(* IEC 61131-3 sources: drain_system/build, 2 files *)

(* ---- plc.st ---- *)
TYPE
  LOGLEVEL : (CRITICAL, WARNING, INFO, DEBUG) := INFO;
END_TYPE

FUNCTION_BLOCK LOGGER
  VAR_INPUT
    TRIG : BOOL;
    MSG : STRING;
    LEVEL : LOGLEVEL := INFO;
  END_VAR
  VAR
    TRIG0 : BOOL;
  END_VAR

  IF TRIG AND NOT TRIG0 THEN
  {{
   LogMessage(GetFbVar(LEVEL),(char*)GetFbVar(MSG, .body),GetFbVar(MSG, .len));
  }}
  END_IF;
  TRIG0:=TRIG;
END_FUNCTION_BLOCK

FUNCTION_BLOCK python_eval
  VAR_INPUT
    TRIG : BOOL;
    CODE : STRING;
  END_VAR
  VAR_OUTPUT
    ACK : BOOL;
    RESULT : STRING;
  END_VAR
  VAR
    STATE : DWORD;
    BUFFER : STRING;
    PREBUFFER : STRING;
    TRIGM1 : BOOL;
    TRIGGED : BOOL;
  END_VAR

  {extern void __PythonEvalFB(int, PYTHON_EVAL*);__PythonEvalFB(0, data__);}
END_FUNCTION_BLOCK

FUNCTION_BLOCK python_poll
  VAR_INPUT
    TRIG : BOOL;
    CODE : STRING;
  END_VAR
  VAR_OUTPUT
    ACK : BOOL;
    RESULT : STRING;
  END_VAR
  VAR
    STATE : DWORD;
    BUFFER : STRING;
    PREBUFFER : STRING;
    TRIGM1 : BOOL;
    TRIGGED : BOOL;
  END_VAR

  {extern void __PythonEvalFB(int, PYTHON_EVAL*);__PythonEvalFB(1,(PYTHON_EVAL*)(void*)data__);}
END_FUNCTION_BLOCK

FUNCTION_BLOCK python_gear
  VAR_INPUT
    N : UINT;
    TRIG : BOOL;
    CODE : STRING;
  END_VAR
  VAR_OUTPUT
    ACK : BOOL;
    RESULT : STRING;
  END_VAR
  VAR
    py_eval : python_eval;
    COUNTER : UINT;
    ADD10_OUT : UINT;
    EQ13_OUT : BOOL;
    SEL15_OUT : UINT;
    AND7_OUT : BOOL;
  END_VAR

  ADD10_OUT := ADD(COUNTER, 1);
  EQ13_OUT := EQ(N, ADD10_OUT);
  SEL15_OUT := SEL(EQ13_OUT, ADD10_OUT, 0);
  COUNTER := SEL15_OUT;
  AND7_OUT := AND(EQ13_OUT, TRIG);
  py_eval(TRIG := AND7_OUT, CODE := CODE);
  ACK := py_eval.ACK;
  RESULT := py_eval.RESULT;
END_FUNCTION_BLOCK

PROGRAM PLC_Drain_System
  VAR
    X_Sensor_ON : BOOL;
  END_VAR
  VAR
    C_Timer : BOOL;
    C_Buzer : BOOL;
  END_VAR
  VAR
    Y_Buzer : BOOL;
    Y_Motor : BOOL;
  END_VAR
  VAR
    Delay : TIME := T#1S;
    TP0 : TP;
    TON0 : TON;
  END_VAR

  Y_Motor := X_Sensor_ON;
  TP0(IN := NOT(C_Timer), PT := Delay);
  Y_Buzer := X_Sensor_ON AND TP0.Q;
  C_Buzer := NOT(TP0.Q);
  TON0(IN := C_Buzer AND NOT(C_Timer), PT := Delay);
  C_Timer := TON0.Q;
END_PROGRAM

CONFIGURATION Config0

  RESOURCE Res0 ON PLC
    TASK task0(INTERVAL := T#20ms,PRIORITY := 0);
    PROGRAM instance0 WITH task0 : PLC_Drain_System;
  END_RESOURCE
END_CONFIGURATION

(* ---- generated_plc.st ---- *)
PROGRAM PLC_Drain_System
  VAR
    X_Sensor_ON AT %IX0.1 : BOOL;
  END_VAR
  VAR
    C_Timer : BOOL;
    C_Buzer : BOOL;
  END_VAR
  VAR
    Y_Buzer AT %QX0.1 : BOOL;
    Y_Motor AT %QX0.2 : BOOL;
  END_VAR
  VAR
    Delay : TIME := T#1S;
    TP0 : TP;
    TON0 : TON;
  END_VAR

  Y_Motor := X_Sensor_ON;
  TP0(IN := NOT(C_Timer), PT := Delay);
  Y_Buzer := X_Sensor_ON AND TP0.Q;
  C_Buzer := NOT(TP0.Q);
  TON0(IN := C_Buzer AND NOT(C_Timer), PT := Delay);
  C_Timer := TON0.Q;
END_PROGRAM

CONFIGURATION Config0

  RESOURCE Res0 ON PLC
    TASK task0(INTERVAL := T#20ms,PRIORITY := 0);
    PROGRAM instance0 WITH task0 : PLC_Drain_System;
  END_RESOURCE
END_CONFIGURATION
